// TwinCAT 3 PLC project PlcIotMqttSampleUsingCallback
// ProgramVersion: 3.1.4020.4
// libraries:
//   Tc2_Standard, * (Beckhoff Automation GmbH)
//   Tc2_System, * (Beckhoff Automation GmbH)
//   Tc2_Utilities, * (Beckhoff Automation GmbH)
//   Tc3_IotBase, * (Beckhoff Automation GmbH)
//   Tc3_Module, * (Beckhoff Automation GmbH)
// project tree:
//   / PlcTask.TcTTO
//   POUs/ FB_MyMqtt.TcPOU, MAIN.TcPOU (not stored), PrgMqttCom.TcPOU
// real-time tasks:
//   TASK PlcTask: cycle T#10ms, priority 20, ADS port 350

CONFIGURATION PlcIotMqttSampleUsingCallback
    RESOURCE PLC ON TwinCAT3
        TASK PlcTask(INTERVAL := T#10ms, PRIORITY := 20);
        PROGRAM MAIN WITH PlcTask : MAIN;
    END_RESOURCE
END_CONFIGURATION

// ---- POUs/FB_MyMqtt.TcPOU
{attribute 'c++_compatible'}
FUNCTION_BLOCK FB_MyMqtt EXTENDS FB_IotMqttClient
VAR_INPUT
END_VAR
VAR_OUTPUT
END_VAR

VAR
	(* received message *)
	{attribute 'TcEncoding':='UTF-8'}
	sTopicRcv : STRING(255);
	{attribute 'TcEncoding':='UTF-8'}
	sPayloadRcv : STRING(255);
END_VAR

{attribute 'c++_compatible'}
{attribute 'pack_mode' := '4'}
{attribute 'show'}
{attribute 'minimal_input_size' := '4'}
METHOD OnMqttMessage : HRESULT
VAR_IN_OUT CONSTANT
	topic	: STRING;
END_VAR
VAR_INPUT
	payload	: PVOID;
	length	: UDINT;
	qos	: TcIotMqttQos;
	repeated	: BOOL;
END_VAR

VAR
	nPayloadRcvLen : UDINT;
END_VAR
SUPER^.nMessagesRcv := SUPER^.nMessagesRcv + 1;

STRNCPY( ADR(sTopicRcv), ADR(topic), SIZEOF(sTopicRcv) );             // important to use STRNCPY() to avoid an access to non-allocated memory
nPayloadRcvLen := MIN(length, DINT_TO_UDINT(SIZEOF(sPayloadRcv))-1);
MEMCPY( ADR(sPayloadRcv), payload, nPayloadRcvLen );
sPayloadRcv[nPayloadRcvLen] := 0;                                     // ensure a null termination of received string

OnMqttMessage := S_OK;
END_METHOD

END_FUNCTION_BLOCK

// ---- POUs/PrgMqttCom.TcPOU
PROGRAM PrgMqttCom
VAR
	fbMqttClient : FB_MyMqtt;
	bSetParameter : BOOL := TRUE;
	bConnect : BOOL := TRUE;
	
	(* published message *)
	sTopicPub : STRING(255) := 'MyTopic';
	sPayloadPub : STRING(255);
	i: UDINT;
	fbTimer : TON := (PT:=T#1S);
	
	bSubscribed : BOOL;
	sTopicSub : STRING(255) := 'MyTopic';
	
	hrErrorOccurred : HRESULT; // contains the latest occurred error
END_VAR

IF bSetParameter THEN
	bSetParameter := FALSE;
	fbMqttClient.sHostName:= 'localhost';
	fbMqttClient.nHostPort:= 1883;
//	fbMqttClient.sClientId:= 'MyTcMqttClient'; 
	fbMqttClient.sTopicPrefix:= ''; 
//	fbMqttClient.nKeepAlive:= 60; 
//	fbMqttClient.sUserName:= ;
//	fbMqttClient.sUserPassword:= ; 
//	fbMqttClient.stWill:= ; 
//	fbMqttClient.stTLS:= ;
END_IF

fbMqttClient.Execute(bConnect);
IF fbMqttClient.bError THEN
	// add your error logging here
	hrErrorOccurred := fbMqttClient.hrErrorCode;
END_IF

IF fbMqttClient.bConnected THEN
	IF NOT bSubscribed THEN
		bSubscribed := fbMqttClient.Subscribe(sTopic:=sTopicSub, eQoS:=TcIotMqttQos.AtMostOnceDelivery);
		IF fbMqttClient.bError THEN
			// add your error logging here
			hrErrorOccurred := fbMqttClient.hrErrorCode;
		END_IF
	END_IF
	fbTimer(IN:=TRUE);
	IF fbTimer.Q THEN // publish new payload every second
		fbTimer(IN:=FALSE);
		i := i + 1;
		sPayloadPub := CONCAT('MyMessage', TO_STRING(i));
		fbMqttClient.Publish(	sTopic:= sTopicPub, 
								pPayload:= ADR(sPayloadPub), nPayloadSize:= LEN2(ADR(sPayloadPub))+1, 
								eQoS:= TcIotMqttQos.AtMostOnceDelivery, bRetain:= FALSE, bQueue:= FALSE );
		IF fbMqttClient.bError THEN
			// add your error logging here
			hrErrorOccurred := fbMqttClient.hrErrorCode;
		END_IF
	END_IF
END_IF

END_PROGRAM
